// TIA Portal V17 export
// export: Created 2026-04-12T10:31:20.0606921Z, ExportSetting WithDefaults, DisplayName Totally Integrated Automation Portal, DisplayVersion V17 Update 4, DisplayName TIA Portal Openness, DisplayVersion V17 Update 4, DisplayName TIA Portal Version Control Interface, DisplayVersion V17, DisplayName SINAMICS Startdrive Advanced, DisplayVersion V17, DisplayName SINAMICS Startdrive G130, G150, S120, S150, SINAMICS MV, S210, DisplayVersion V17, DisplayName SINAMICS Startdrive G110M, G120, G120C, G120D, G120P, G115D, DisplayVersion V17, DisplayName STEP 7 Professional, DisplayVersion V17 Update 4, DisplayName STEP 7 Safety, DisplayVersion V17, DisplayName WinCC Advanced, DisplayVersion V17 Update 4
FUNCTION "风机燃气" : Void   // FC3, LAD
{ S7_Optimized_Access := 'TRUE' }
VERSION : 0.1
// stored: AutoNumber true, IsIECCheckEnabled false, SetENOAutomatically false, UDAEnableTagReadback false
   VAR_TEMP   // added for the SCL form of the ladder/FBD networks
      _w1 : Bool;
   END_VAR
BEGIN

REGION Network 1: 风机输出
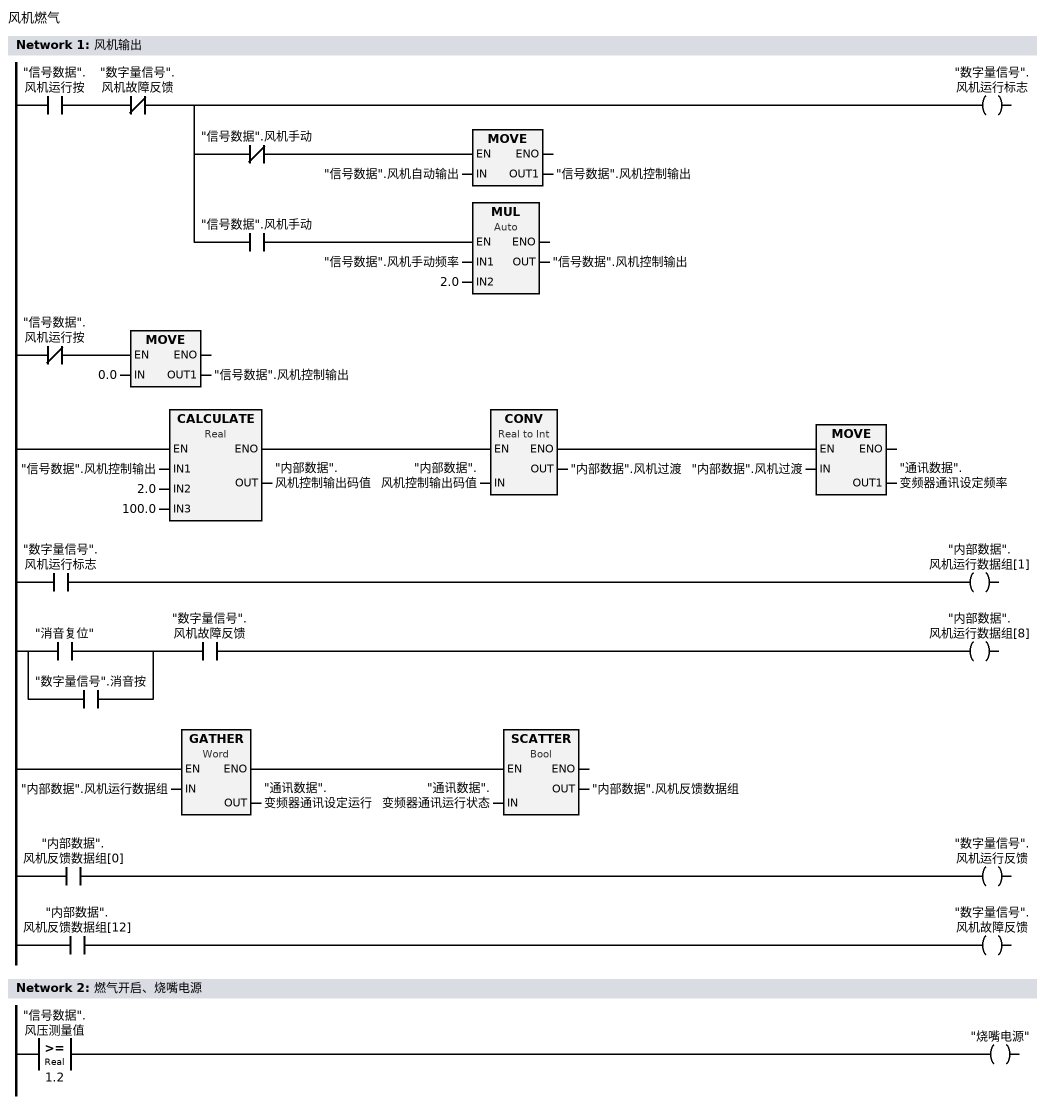
   RUNG wire#powerrail
      Contact( "信号数据".风机运行按 )
      I_Contact( "数字量信号".风机故障反馈 )
      wire#w1
      Coil( "数字量信号".风机运行标志 )
   END_RUNG
   RUNG wire#w1
      I_Contact( "信号数据".风机手动 )
      Move(in := "信号数据".风机自动输出, out1 => "信号数据".风机控制输出)
   END_RUNG
   RUNG wire#w1
      Contact( "信号数据".风机手动 )
      Mul(in1 := "信号数据".风机手动频率, in2 := 2.0, out => "信号数据".风机控制输出)
   END_RUNG
   RUNG wire#powerrail
      I_Contact( "信号数据".风机运行按 )
      Move(in := 0.0, out1 => "信号数据".风机控制输出)
   END_RUNG
   RUNG wire#powerrail
      { S7_Templates := "SrcType := Real"; S7_Expression := "(IN1/IN2)*IN3" } Calculate(in1 := "信号数据".风机控制输出, in2 := 2.0, in3 := 100.0, out => "内部数据".风机控制输出码值)
      { S7_Templates := "[SrcType := Real, DestType := Int]" } Convert(in := "内部数据".风机控制输出码值, out => "内部数据".风机过渡)
      Move(in := "内部数据".风机过渡, out1 => "通讯数据".变频器通讯设定频率)
   END_RUNG
   RUNG wire#powerrail
      Contact( "数字量信号".风机运行标志 )
      Coil( "内部数据".风机运行数据组[1] )
   END_RUNG
   RUNG wire#powerrail
      Contact( "消音复位" )
      wire#w2
      Contact( "数字量信号".风机故障反馈 )
      Coil( "内部数据".风机运行数据组[8] )
   END_RUNG
   RUNG wire#powerrail
      Contact( "数字量信号".消音按 )
   END_RUNG wire#w2
   RUNG wire#powerrail
      { S7_Templates := "[dest_type := Word, src_type := Bool]" } GATHER(IN := "内部数据".风机运行数据组, OUT => "通讯数据".变频器通讯设定运行)
      { S7_Templates := "[dest_type := Bool, src_type := Word]" } SCATTER(IN := "通讯数据".变频器通讯运行状态, OUT => "内部数据".风机反馈数据组)
   END_RUNG
   RUNG wire#powerrail
      Contact( "内部数据".风机反馈数据组[0] )
      Coil( "数字量信号".风机运行反馈 )
   END_RUNG
   RUNG wire#powerrail
      Contact( "内部数据".风机反馈数据组[12] )
      Coil( "数字量信号".风机故障反馈 )
   END_RUNG
   // the same network as SCL:
   "数字量信号".风机运行标志 := "信号数据".风机运行按 AND NOT "数字量信号".风机故障反馈;
   IF "数字量信号".风机运行标志 AND NOT "信号数据".风机手动 THEN "信号数据".风机控制输出 := "信号数据".风机自动输出; END_IF;
   IF "数字量信号".风机运行标志 AND "信号数据".风机手动 THEN "信号数据".风机控制输出 := "信号数据".风机手动频率 * 2.0; END_IF;
   IF NOT "信号数据".风机运行按 THEN "信号数据".风机控制输出 := 0.0; END_IF;
   "内部数据".风机控制输出码值 := ("信号数据".风机控制输出/2.0)*100.0;
   "内部数据".风机过渡 := REAL_TO_INT("内部数据".风机控制输出码值);
   "通讯数据".变频器通讯设定频率 := "内部数据".风机过渡;
   "内部数据".风机运行数据组[1] := "数字量信号".风机运行标志;
   "内部数据".风机运行数据组[8] := ("消音复位" OR "数字量信号".消音按) AND "数字量信号".风机故障反馈;
   GATHER(IN := "内部数据".风机运行数据组, OUT => "通讯数据".变频器通讯设定运行, ENO => #_w1);
   IF #_w1 THEN SCATTER(IN := "通讯数据".变频器通讯运行状态, OUT => "内部数据".风机反馈数据组); END_IF;
   "数字量信号".风机运行反馈 := "内部数据".风机反馈数据组[0];
   "数字量信号".风机故障反馈 := "内部数据".风机反馈数据组[12];
END_REGION

REGION Network 2: 燃气开启、烧嘴电源
   RUNG wire#powerrail
      { S7_Templates := "SrcType := Real" } GE_Contact(in1 := "信号数据".风压测量值, in2 := 1.2)
      Coil( "烧嘴电源" )
   END_RUNG
   // the same network as SCL:
   "烧嘴电源" := "信号数据".风压测量值 >= 1.2;
END_REGION
END_FUNCTION
